TYPE
    ST_MessageBox_Response : STRUCT
        ErrorRaised      : BOOL;
        ErrorAcknowledge : BOOL;
        ErrorSolution    : USINT;
    END_STRUCT
END_TYPE

(* stored: Version 1.1.0.1
   DUT ST_MessageBox_Response: Id {a62e7db7-6278-488d-ac33-64b03a299723} *)
